FUNCTION_BLOCK FB_Property IMPLEMENTS I_Property
VAR_INPUT
END_VAR
VAR_OUTPUT
END_VAR
VAR
	fbStringBuilder:	FB_StringBuilder;
	fbList:				FB_ListSTRING;
END_VAR

METHOD PUBLIC M_Add : BOOL
VAR_INPUT
	Name:			STRING(255);
	Value:			STRING(255);
END_VAR
VAR
	nIndex: 		INT;
	sKey:			STRING(255);
END_VAR
fbStringBuilder.M_Reset();
fbStringBuilder.M_Append('<property name="');
fbStringBuilder.M_Append(Name);
sKey:= fbStringBuilder.M_ToString();
fbStringBuilder.M_Append('" value="');
fbStringBuilder.M_Append(Value);
fbStringBuilder.M_Append('" />');

WHILE nIndex < fbList.P_Length DO
	IF FIND(fbList.M_Item(nIndex), sKey) <> 0 THEN
		fbList.M_Set(nIndex, fbStringBuilder.M_ToString());
		RETURN;
	END_IF
	nIndex:= nIndex +1;
END_WHILE
fbList.M_Add(fbStringBuilder.M_ToString());
M_Add:= TRUE;
END_METHOD

METHOD PUBLIC M_Reset
fbStringBuilder.M_Reset();
fbList.M_Clear();
END_METHOD

PROPERTY PUBLIC P_List : I_ListSTRING
GET
P_List:= fbList;
END_GET
END_PROPERTY

END_FUNCTION_BLOCK

(* stored: Version 1.1.0.1
   POU FB_Property: Id {9f663162-7495-088d-0f62-2a9bab2c599e}, SpecialFunc None
   Method M_Add: Id {a2860717-79b0-0674-3a4b-10a52016875b}
   Method M_Reset: Id {eddb6b8d-8e19-018a-029c-46c6dc54bfcd}
   Property P_List: Id {9de6c82c-01dc-0311-3188-815453a357f8}
   Get Get: Id {82c776c2-c9a9-06fc-1a5f-e6c70e7b25b9} *)
